FUNCTION_BLOCK PUBLIC FB_Conv1
VAR_INPUT
END_VAR
VAR_OUTPUT
END_VAR
VAR
	Timer1				:	TON	;
	x					: INT :=0;
	Set_Motor			:	BOOL;
	Reset_Motor			:	BOOL;	
	iSTEP				:	INT;
END_VAR

CASE iSTEP OF 
	
	// ================================================  Conveyor Motor n Re Cyl Init
	0:	IF IO.bConv_Ready AND IO_control.bEstop THEN
			IO_control.bMotor1 := FALSE;
			IO_control.bReCyl_Ext := TRUE ;
			IO_control.bReCyl_Ret := FALSE ;
			IF IO.bReCyl1_State_Extend THEN
				iSTEP := 2 ;
			END_IF
		END_IF

	// ================================================  wait for bin,,,.... fbdroptask/fbdropoff will run in d background	
	2:	IF IO_Conveyor.bReceiving_Complete AND IO.bConv1_In THEN
			IF IO_Conveyor.bExit1_IsOpen THEN
				iSTEP := iSTEP + 1 ;
			END_IF	
		END_IF
	
	// ================================================  Receiving cyl to retract after receiving complete
	3:	IO_Conveyor.bExit1_IsOpen := FALSE;
		IO_control.bReCyl_Ext := FALSE ;
		IO_control.bReCyl_Ret := TRUE ;
		IO_Conveyor.bReceiving_Complete := FALSE;
		IF IO.bReCyl1_State_Retract THEN
			IO.bPoatman_get := TRUE;
			IO_Conveyor.bReCylinder_At_Work := FALSE;				
			iSTEP := iSTEP + 1 ;
		ELSE
			IO_Conveyor.bReCylinder_At_Work := TRUE;
		END_IF
	
	// ================================================  motor start after re cyl retract	
	4:	Timer1(IN:= NOT IO_Conveyor.bReCylinder_At_Work, PT:=T#0.1S, Q=> Set_Motor);
		IO_control.bMotor1 S= Set_Motor;
		IF Set_Motor THEN
			IO.bPoatman_get := FALSE;
			iSTEP := iSTEP + 1 ;
		END_IF	
	
	// ================================================  stop motor1 if conv1_out ON	
	5: 	IF IO.bConv1_Out THEN
			IO_control.bReCyl_Ext := TRUE;
			IO_control.bReCyl_Ret := FALSE;
			IO_Conveyor.Bin_At_Exit_1 := TRUE;
			IO_control.bMotor1 R= IO.bConv1_Out;
			iSTEP := iSTEP + 1;
		END_IF

	// ================================================  update status for conv1 job done
	6:	IO_Conveyor.Conv1_Done := TRUE;
		iSTEP := iSTEP + 1;
	
	// ================================================  receive feedback from conv2
	(*receive reset for conv1 job done*)
	7:	IF NOT IO_Conveyor.Conv1_Done THEN
			IO_Conveyor.Bin_At_Exit_1 := FALSE;
			iSTEP := 0;
		END_IF							
END_CASE

IF IO.bManualMode OR IO.bEstop_State THEN
	IO_Conveyor.Bin_At_Exit_1 := FALSE;
	IO_Conveyor.Conv1_Done := FALSE;
	IO_Conveyor.Bin_At_Exit_1 := FALSE;
	IO.bPoatman_get := FALSE;
	IO_Conveyor.bReCylinder_At_Work := FALSE;
	FOR x := 1 TO 8 DO
		IO.abinID_Set[x] := '';
	END_FOR
	iSTEP := 0 ;
END_IF

END_FUNCTION_BLOCK

(* stored: Version 1.1.0.1, ProductVersion 3.1.4024.12
   POU FB_Conv1: Id {69996449-2c84-4955-a424-7766fe39a2d2}, SpecialFunc None *)
